TYPE ST_RecStatus ://纠偏系统
STRUCT
    bError             :BOOL;     //纠偏故障
    bRuning           :BOOL;    //纠偏运行中
END_STRUCT
END_TYPE

(* stored: Version 1.1.0.1, ProductVersion 3.1.4024.9
   DUT ST_RecStatus: Id {3e872998-4d7d-4ce4-903a-12e6bf235113} *)
